(* IEC 61131-3 sources: CodesysTest/export/UN00 - Sharp Bagger/EM01 - Bagger Head/CM00 - Bag Open Fingers/Base/Tests/FB_BaseBagOpenFingers_UnitTest.pou, 2 files *)

(* ---- FB_BaseBagOpenFingers_UnitTest.pou.st ---- *)
(*#-#-#-#-#-#-#-#-#-#---Declaration---#-#-#-#-#-#-#-#-#-#-#-#-#*)

{attribute 'test' := 'multitest'}
{attribute 'testcasename':='Base Bag Open Fingers'}
{attribute 'testcategory':='Machine Components'}
{attribute 'testcasetimeout':='5000'}

FUNCTION_BLOCK FB_BaseBagOpenFingers_UnitTest EXTENDS CBM.EtrigA
VAR_INPUT
	xGetTestInfo : BOOL;
    diTestCaseIndex : DINT;
END_VAR
VAR_OUTPUT
    sTestCaseName : STRING;
	sTestCaseCategories : STRING;
    diTestCaseCount : DINT;
    diTestCaseTimeout : DINT;
    sInfo : STRING;
	eError : UnitTestErrors;
    sError : STRING;
    eFailureMode : TM.FAILUREMODE;
END_VAR
VAR
	testee : FB_BaseBagOpenFingers(name := 'Test Base Bag Open Fingers');
	checkGrabTimer : Standard.TON;
	checkNotGrabTimer : Standard.TON;
	grabRequested : BOOL;
END_VAR
(*#-#-#-#-#-#-#-#-#-#---Implementation---#-#-#-#-#-#-#-#-#-#-#-#-#*)

SUPER^();

(* ---- prvCyclicAction.m.st ---- *)
(*#-#-#-#-#-#-#-#-#-#---Declaration---#-#-#-#-#-#-#-#-#-#-#-#-#*)

{attribute 'hide'}
METHOD prvCyclicAction : BOOL
(*#-#-#-#-#-#-#-#-#-#---Implementation---#-#-#-#-#-#-#-#-#-#-#-#-#*)

SUPER^.prvCyclicAction();
checkGrabTimer();
checkNotGrabTimer();
testee(
	delayToGrabSetting:= ,
	delayToCheckBagPresentSetting:= ,
	delayToClearSetting:= ,
	grabCounter=> ,
	releaseCounter=> ,
	missedCounter=> );
CASE diTestCaseIndex OF
    0: 	IF THIS^.xGetTestInfo THEN
            THIS^.sTestCaseName := 'Step 1: Check all statuses are clear on initialization';
            THIS^.sTestCaseCategories := 'Machine Components';
            THIS^.diTestCaseTimeout := 3000;
			xDone := TRUE;
		ELSE
			IF NOT testee.BagCleared
				AND NOT testee.BagGrabbed
				AND NOT testee.BagMissed
			THEN
				 xDone := TRUE;
			ELSE
				THIS^.sError := 'Status should be all false';
				xError := TRUE;
				eError := UnitTestErrors.Failure;
            	eFailureMode := TM.FAILUREMODE.AbortTestCase;
                iError := 1;
			END_IF
        END_IF
    1: 	IF THIS^.xGetTestInfo THEN
            THIS^.sTestCaseName := 'Step 2: Grab Bag and watch for BagGrabbed status';
            THIS^.sTestCaseCategories := 'Machine Components';
            THIS^.diTestCaseTimeout := 3000;
			xDone := TRUE;
		ELSE
			testee.delayToGrabSetting := 1.0;
			checkGrabTimer.IN := TRUE;
			checkGrabTimer.PT := T#1050MS;

			checkNotGrabTimer.IN := TRUE;
			checkNotGrabTimer.PT := T#900MS;

			IF NOT grabRequested THEN
				testee.GrabBag();
				grabRequested := TRUE;
			END_IF

			IF checkNotGrabTimer.Q THEN
				IF testee.delayToGrab.Q THEN
					THIS^.sError := 'Bag Grab Request occured too soon';
					xError := TRUE;
					eError := UnitTestErrors.Failure;
					eFailureMode := TM.FAILUREMODE.AbortTestCase;
					iError := 1;
				END_IF
				checkNotGrabTimer.IN := FALSE;
			ELSIF checkGrabTimer.Q THEN
				IF testee.delayToGrab.Q THEN
					xDone := TRUE;
				ELSE
					THIS^.sError := 'Bag Grab Timer not timed out';
					xError := TRUE;
					eError := UnitTestErrors.Failure;
					eFailureMode := TM.FAILUREMODE.AbortTestCase;
					iError := 1;
				END_IF
				checkGrabTimer.IN := FALSE;
			END_IF
        END_IF

    ELSE
        IF THIS^.diTestCaseIndex < 0 THEN
            THIS^.diTestCaseCount := 2;
            xDone := TRUE;
        ELSE
            THIS^.sInfo := 'Invalid test case index';
            eError := UnitTestErrors.Failure;
			xError := TRUE;
        END_IF
END_CASE
